// Mitsubishi GX Developer project: 15-1202   PLC: FX3G

PROGRAM MAIN
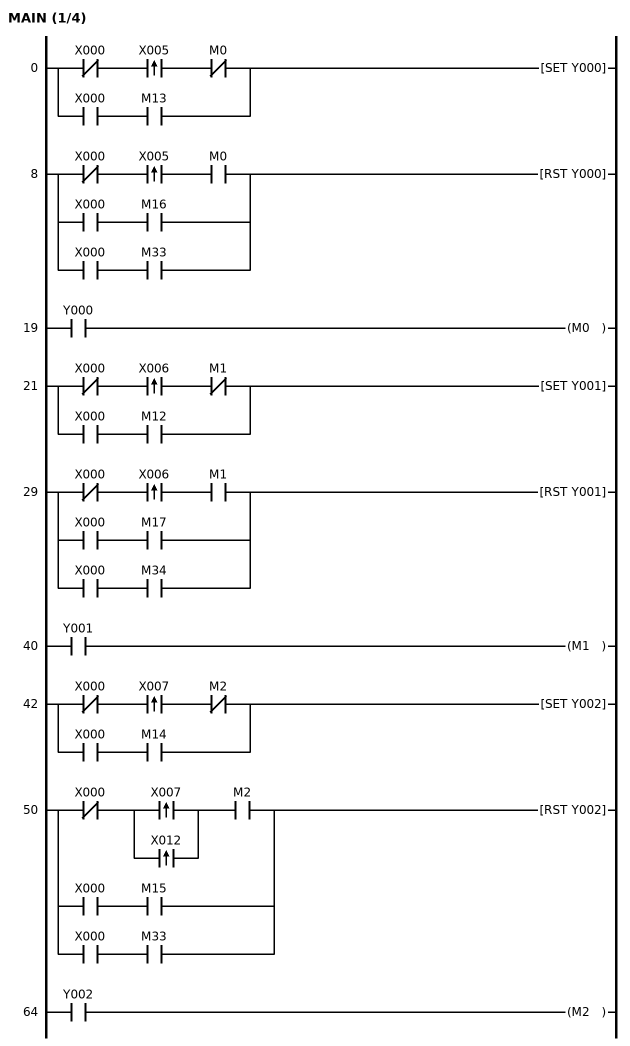
0     LDI     X000
      ANDP    X005
      ANI     M0
      LD      X000
      AND     M13
      ORB
      SET     Y000
8     LDI     X000
      ANDP    X005
      AND     M0
      LD      X000
      AND     M16
      ORB
      LD      X000
      AND     M33
      ORB
      RST     Y000
19    LD      Y000
      OUT     M0
21    LDI     X000
      ANDP    X006
      ANI     M1
      LD      X000
      AND     M12
      ORB
      SET     Y001
29    LDI     X000
      ANDP    X006
      AND     M1
      LD      X000
      AND     M17
      ORB
      LD      X000
      AND     M34
      ORB
      RST     Y001
40    LD      Y001
      OUT     M1
42    LDI     X000
      ANDP    X007
      ANI     M2
      LD      X000
      AND     M14
      ORB
      SET     Y002
50    LDI     X000
      LDP     X007
      ORP     X012
      ANB
      AND     M2
      LD      X000
      AND     M15
      ORB
      LD      X000
      AND     M33
      ORB
      RST     Y002
64    LD      Y002
      OUT     M2
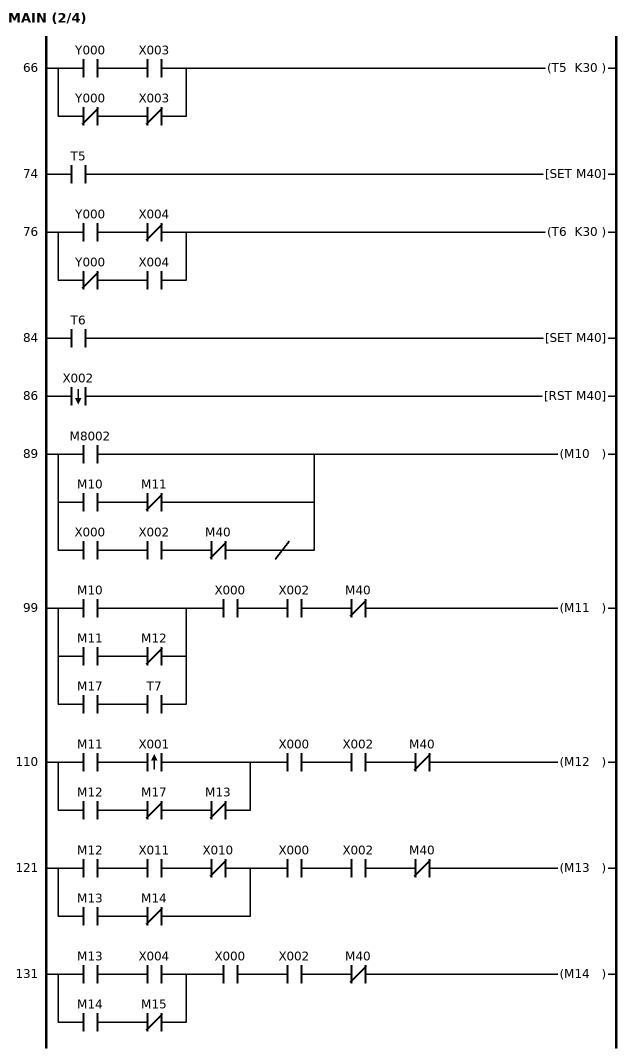
66    LD      Y000
      AND     X003
      LDI     Y000
      ANI     X003
      ORB
      OUT     T5 K30
74    LD      T5
      SET     M40
76    LD      Y000
      ANI     X004
      LDI     Y000
      AND     X004
      ORB
      OUT     T6 K30
84    LD      T6
      SET     M40
86    LDF     X002
      RST     M40
89    LD      M8002
      LD      M10
      ANI     M11
      ORB
      LD      X000
      AND     X002
      ANI     M40
      INV
      ORB
      OUT     M10
99    LD      M10
      LD      M11
      ANI     M12
      ORB
      LD      M17
      AND     T7
      ORB
      AND     X000
      AND     X002
      ANI     M40
      OUT     M11
110   LD      M11
      ANDP    X001
      LD      M12
      ANI     M17
      ANI     M13
      ORB
      AND     X000
      AND     X002
      ANI     M40
      OUT     M12
121   LD      M12
      AND     X011
      ANI     X010
      LD      M13
      ANI     M14
      ORB
      AND     X000
      AND     X002
      ANI     M40
      OUT     M13
131   LD      M13
      AND     X004
      LD      M14
      ANI     M15
      ORB
      AND     X000
      AND     X002
      ANI     M40
      OUT     M14
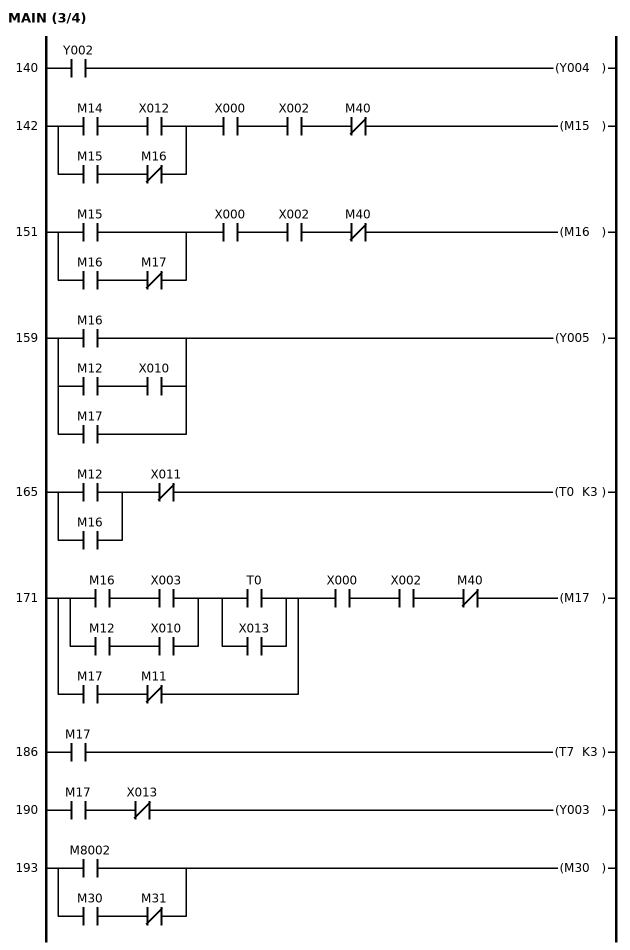
140   LD      Y002
      OUT     Y004
142   LD      M14
      AND     X012
      LD      M15
      ANI     M16
      ORB
      AND     X000
      AND     X002
      ANI     M40
      OUT     M15
151   LD      M15
      LD      M16
      ANI     M17
      ORB
      AND     X000
      AND     X002
      ANI     M40
      OUT     M16
159   LD      M16
      LD      M12
      AND     X010
      ORB
      OR      M17
      OUT     Y005
165   LD      M12
      OR      M16
      ANI     X011
      OUT     T0 K3
171   LD      M16
      AND     X003
      LD      M12
      AND     X010
      ORB
      LD      T0
      OR      X013
      ANB
      LD      M17
      ANI     M11
      ORB
      AND     X000
      AND     X002
      ANI     M40
      OUT     M17
186   LD      M17
      OUT     T7 K3
190   LD      M17
      ANI     X013
      OUT     Y003
193   LD      M8002
      LD      M30
      ANI     M31
      ORB
      OUT     M30
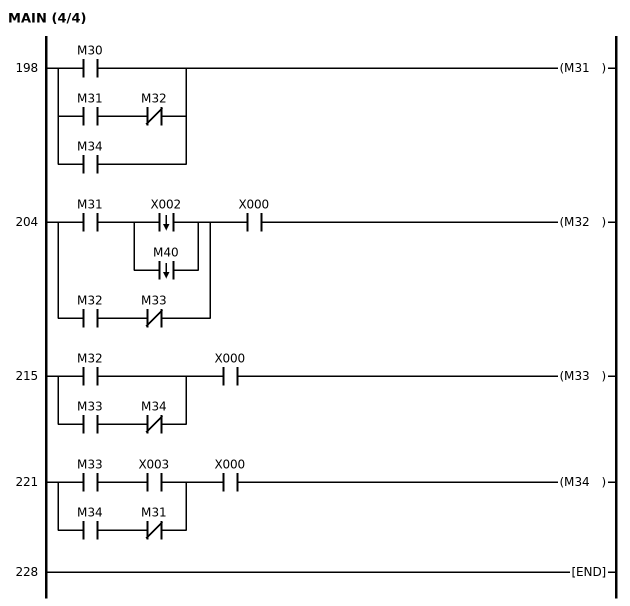
198   LD      M30
      LD      M31
      ANI     M32
      ORB
      OR      M34
      OUT     M31
204   LD      M31
      LDF     X002
      ORF     M40
      ANB
      LD      M32
      ANI     M33
      ORB
      AND     X000
      OUT     M32
215   LD      M32
      LD      M33
      ANI     M34
      ORB
      AND     X000
      OUT     M33
221   LD      M33
      AND     X003
      LD      M34
      ANI     M31
      ORB
      AND     X000
      OUT     M34
228   END
END_PROGRAM
